Staubli VAL3: removeAction.pgx

public program removeAction()
begin
  // mutex it
  setMutex(bActionMutex)
  // remove the action
  if size(aAction)>1
    delete(aAction[0])
  else
    // remove
    resize(aAction[0].iInstr,1,1)
    aAction[0].iInstr.sType="null"
    aAction[0].iInstr.sData=""
    aAction.nPointId=0
  endIf
  // release
  bActionMutex=false
end
